{attribute 'GeneratedUsingTerminal: EL5001--0000'}
{attribute addProperty BoxType "EL5001--0000"}
{attribute addProperty Id "Channel_1AT %I*Channel_4E63E14D5WcStateAT %I*WcState_9091E0EB2InfoDataAT %I*InfoData_94A18F5E2"}
{attribute addProperty CRC "1102484513"}
{attribute addProperty Size "9"}
TYPE EL5001_41B69421 EXTENDS EtcSlaveTerminalBase_947E5A46 :
STRUCT
	{attribute addProperty Name "Channel_1"}
	Channel_1 : Channel_4E63E14D;
	{attribute addProperty Name "WcState"}
	WcState : WcState_9091E0EB;
	{attribute addProperty Name "InfoData"}
	InfoData : InfoData_94A18F5E;
END_STRUCT
END_TYPE

(* stored: Version 1.2.0.0, ProductVersion 3.1.4024.9
   DUT EL5001_41B69421: Id {8efd453c-19bd-4b86-b175-e140b3431f13} *)
